% RSLogix 500 project PROC1_TIMERS_BAK005.RSS, saved by version 8.30.00.16 %
PROJECT "PROC1"    % processor: Bul.1763 MicroLogix 1100 Series B %

PROGRAM FILES
  LAD 2 "MAIN"  2 rungs
  LAD 3 "TIMERS"  5 rungs  % Various Timer controls %

DATA FILES
  O0 OUTPUT  4 elements
  I1 INPUT  6 elements
  S2 STATUS  66 elements
  B3 BINARY  1 elements
  T4 TIMER  1 elements
  C5 COUNTER  1 elements
  R6 CONTROL  1 elements
  N7 INTEGER  1 elements
  F8 FLOAT  1 elements

LADDER 2 "MAIN"
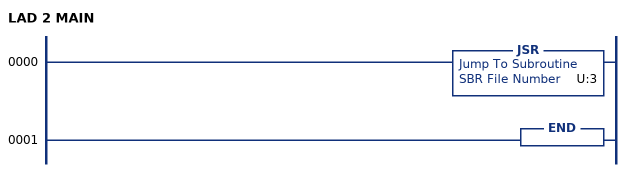
% Rung: 0 %
SOR JSR U:3 EOR
% Rung: 1 %
SOR END EOR

LADDER 3 "TIMERS"    % Various Timer controls %
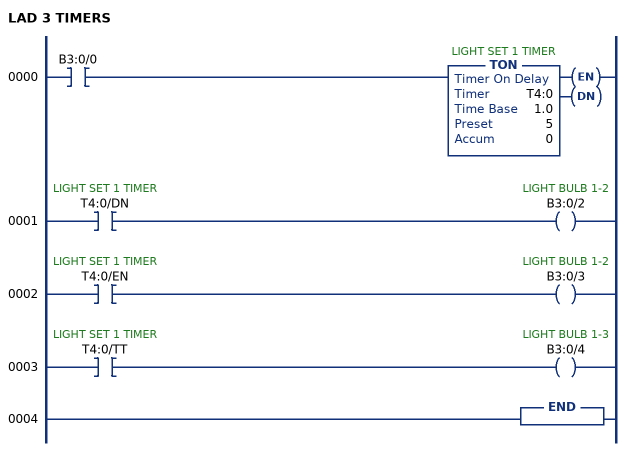
% Rung: 0 %
SOR XIC B3:0/0 TON T4:0 1.0 5 0 EOR
%   T4:0  "LIGHT SET 1 TIMER" %
% Rung: 1 %
SOR XIC T4:0/DN OTE B3:0/2 EOR
%   T4:0  "LIGHT SET 1 TIMER" %
%   B3:0/2  "LIGHT BULB 1-2" %
% Rung: 2 %
SOR XIC T4:0/EN OTE B3:0/3 EOR
%   T4:0  "LIGHT SET 1 TIMER" %
%   B3:0/3  "LIGHT BULB 1-2" %
% Rung: 3 %
SOR XIC T4:0/TT OTE B3:0/4 EOR
%   T4:0  "LIGHT SET 1 TIMER" %
%   B3:0/4  "LIGHT BULB 1-3" %
% Rung: 4 %
SOR END EOR

OTHER DOCUMENTED ADDRESSES
  B3:0  "LIGHT SWITCH 1"
  B3:4  "LIGHT BULB 1-3"

REVISION NOTES
  0: Added LIGHT BULB 1-2
  1: Added LIGHT BULB 1-3
  2: Fixed error
  3: Changed SCAN time to 61 microsecs

DATA TABLE (non-zero values as saved)
DATA T4
% .PRE .ACC %
% T4:0 % 5 0
